// TwinCAT 3 PLC project SerialCom
// ProgramVersion: 3.1.4026.12
// libraries:
//   Tc2_ModbusRTU, * (Beckhoff Automation GmbH)
//   Tc2_SerialCom, * (Beckhoff Automation GmbH)
//   Tc2_Standard, * (Beckhoff Automation GmbH)
//   Tc2_System, * (Beckhoff Automation GmbH)
// project tree:
//   GVLs/ GVL_SerialCom.TcGVL (not stored)
//   / PlcTask.TcTTO
//   POUs/ MAIN.TcPOU, P_SerialCom.TcPOU
// real-time tasks:
//   TASK PlcTask: cycle T#10ms, priority 20, ADS port 350

CONFIGURATION SerialCom
    RESOURCE PLC ON TwinCAT3
        TASK PlcTask(INTERVAL := T#10ms, PRIORITY := 20);
        PROGRAM MAIN WITH PlcTask : MAIN;
    END_RESOURCE
END_CONFIGURATION

// ---- POUs/MAIN.TcPOU
PROGRAM MAIN
VAR
END_VAR

P_SerialCom();

END_PROGRAM

// ---- POUs/P_SerialCom.TcPOU
PROGRAM P_SerialCom
VAR
	(*テストではパソコンにシリアルポートが無いので未使用
	fbModbusRtuSlave_PcCOM			:ModbusRtuSlave_PcCOM;
	*)
	
	//テスト用のファンクションブロック
	fbSerialLineControlADS				:SerialLineControlADS;
	fbModbusRtuSlave_Generic			:ModbusRtuSlave_Generic;
	
	//テスト用の変数
	bConnect							:BOOL:=TRUE;
	stSerialCfg							:ComSerialConfig;
	RxBuffer							:ComBuffer;
	TxBuffer							:ComBuffer;
	bAdsError							:BOOL;
	nAdsErrorID							:UDINT;	

END_VAR

//----テスト用のModbus通信---
	//シリアル接続を設定
	stSerialCfg.ComPort			:=3;
	stSerialCfg.Baudrate		:=9600;
	stSerialCfg.Parity			:=PARITY_NONE;
	stSerialCfg.DataBits		:=8;
	stSerialCfg.StopBits		:=STOPBITS_ONE;
	stSerialCfg.DTR				:=DTR_CTRL_DISABLE;
	stSerialCfg.RTS				:=RTS_CTRL_DISABLE;
	stSerialCfg.CTS				:=FALSE;
	stSerialCfg.DSR				:=FALSE;
	
	//USB接続のシリアルポートで通信
	fbSerialLineControlADS(	Connect		:=bConnect,
							SerialCfg	:=stSerialCfg,
							NetId		:='192.168.15.15.1.1',
							Timeout		:=DEFAULT_ADS_TIMEOUT,
							TxBuffer	:=TxBuffer,
							RxBuffer	:=RxBuffer,
							PortOpened	=>,
							Error		=>bAdsError,
							ErrorID		=>nAdsErrorID,
							Busy		=>,
							TxBufCount	=>,
							RxBufCount	=>
							);
	
	//Modbus通信
	fbModbusRtuSlave_Generic(	UnitID				:=1,
								AdrInputs			:=ADR(GVL_SerialCom.Inputs),
								SizeInputBytes		:=SIZEOF(GVL_SerialCom.Inputs),
								AdrOutputs			:=ADR(GVL_SerialCom.Outputs),
								SizeOutputBytes		:=SIZEOF(GVL_SerialCom.Outputs),
								AdrMemory			:=ADR(GVL_SerialCom.Memory),
								SizeMemoryBytes		:=SIZEOF(GVL_SerialCom.Memory),
								RxBuffer			:=RxBuffer,
								TxBuffer			:=TxBuffer,
								ErrorId				=>
								);

END_PROGRAM
